% RSLogix 500 project Sauerstoff-Mess- und Kalibriersystem.RSS, saved by version 8.30.00.16 %
PROJECT "UNTITLED"    % processor: Bul.1763 MicroLogix 1100 Series B %

PROGRAM FILES
  LAD 2 "MAIN"  5 rungs
  LAD 3 "IO"  4 rungs
  LAD 4 "KALIBRIERU"  15 rungs

DATA FILES
  O0 OUTPUT  4 elements
  I1 INPUT  6 elements
  S2 STATUS  66 elements
  B3 BINARY  1 elements
  T4 TIMER  4 elements
  C5 COUNTER  1 elements
  R6 CONTROL  1 elements
  N7 INTEGER  9 elements
  F8 FLOAT  6 elements

LADDER 2 "MAIN"
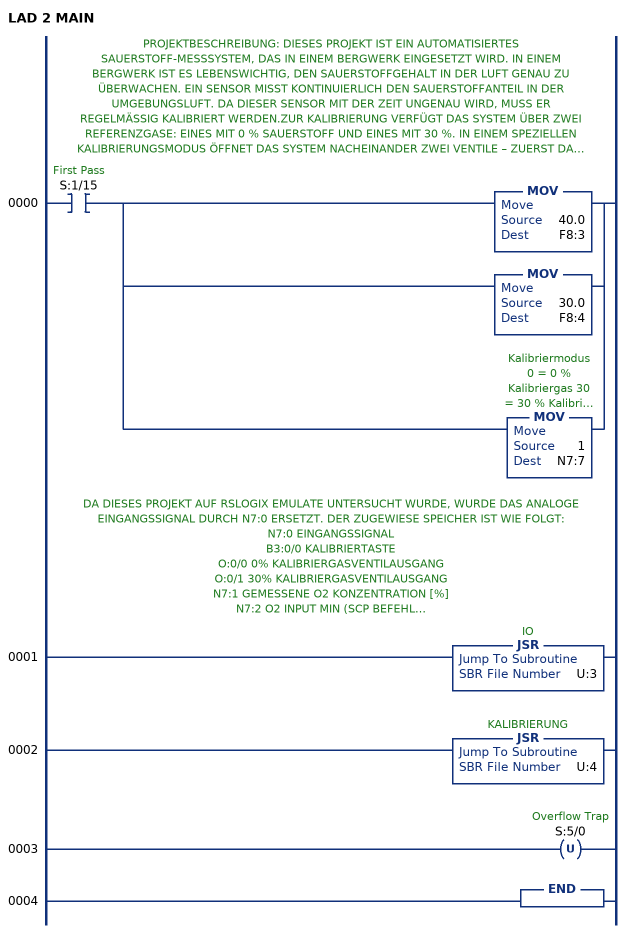
% Rung: 0 %
% PROJEKTBESCHREIBUNG: DIESES PROJEKT IST EIN AUTOMATISIERTES SAUERSTOFF-MESSSYSTEM, DAS IN EINEM BERGWERK EINGESETZT WIRD. IN EINEM BERGWERK IST ES LEBENSWICHTIG, DEN SAUERSTOFFGEHALT IN DER LUFT GENAU ZU ÜBERWACHEN. EIN SENSOR MISST KONTINUIERLICH DEN SAUERSTOFFANTEIL IN DER UMGEBUNGSLUFT. DA DIESER SENSOR MIT DER ZEIT UNGENAU WIRD, MUSS ER REGELMÄSSIG KALIBRIERT WERDEN.ZUR KALIBRIERUNG VERFÜGT DAS SYSTEM ÜBER ZWEI REFERENZGASE: EINES MIT 0 % SAUERSTOFF UND EINES MIT 30 %. IN EINEM SPEZIELLEN KALIBRIERUNGSMODUS ÖFFNET DAS SYSTEM NACHEINANDER ZWEI VENTILE – ZUERST DAS FÜR 0 %-GAS, DANN DAS FÜR 30 %-GAS – UND MISST JEWEILS 30 SEKUNDEN LANG DIE SENSORWERTE. AUS DIESEN MESSUNGEN BERECHNET DAS SYSTEM AUTOMATISCH KORREKTURWERTE, UM SPÄTERE SAUERSTOFFMESSUNGEN WIEDER KORREKT ANZEIGEN ZU KÖNNEN. %
SOR XIC S:1/15 BST MOV 40.0 F8:3 NXB MOV 30.0 F8:4 NXB MOV 1 N7:7 BND EOR
%   S:1/15  "First Pass" %
%   N7:7  "Kalibriermodus 0 = 0 % Kalibriergas 30 = 30 % Kalibriergas 1 = Idle Modus" %
% Rung: 1 %
% DA DIESES PROJEKT AUF RSLOGIX EMULATE UNTERSUCHT WURDE, WURDE DAS ANALOGE EINGANGSSIGNAL DURCH N7:0 ERSETZT. DER ZUGEWIESE SPEICHER IST WIE FOLGT:
% N7:0 EINGANGSSIGNAL
% B3:0/0 KALIBRIERTASTE
% O:0/0 0% KALIBRIERGASVENTILAUSGANG
% O:0/1 30% KALIBRIERGASVENTILAUSGANG
% N7:1 GEMESSENE O2 KONZENTRATION [%]
% N7:2 O2 INPUT MIN (SCP BEFEHL)
% N7:3 O2 INPUT MAX (SCP BEFEHL) %
SOR JSR U:3 EOR
%   U:3  "IO" %
% Rung: 2 %
SOR JSR U:4 EOR
%   U:4  "KALIBRIERUNG" %
% Rung: 3 %
SOR OTU S:5/0 EOR
%   S:5/0  "Overflow Trap" %
% Rung: 4 %
SOR END EOR

LADDER 3 "IO"
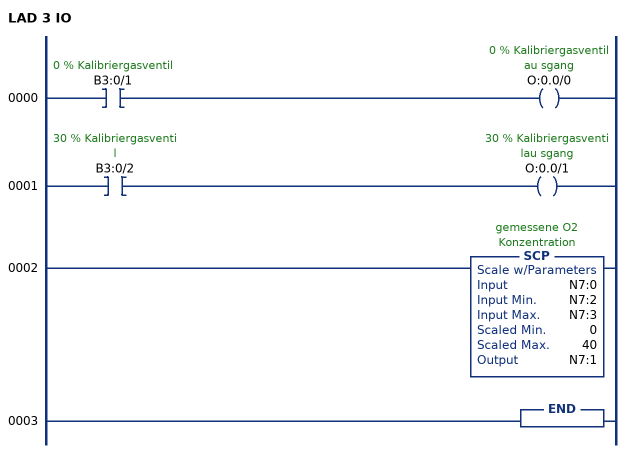
% Rung: 0 %
SOR XIC B3:0/1 OTE O:0.0/0 EOR
%   B3:0/1  "0 % Kalibriergasventil" %
%   O:0.0/0  "0 % Kalibriergasventilau sgang" %
% Rung: 1 %
SOR XIC B3:0/2 OTE O:0.0/1 EOR
%   B3:0/2  "30 % Kalibriergasventil" %
%   O:0.0/1  "30 % Kalibriergasventilau sgang" %
% Rung: 2 %
SOR SCP N7:0 N7:2 N7:3 0 40 N7:1 EOR
%   N7:0  "02 Eingangsignal" %
%   N7:2  "O2 Min" %
%   N7:3  "O2 Max" %
%   N7:1  "gemessene O2 Konzentration" %
% Rung: 3 %
SOR END EOR

LADDER 4 "KALIBRIERU"
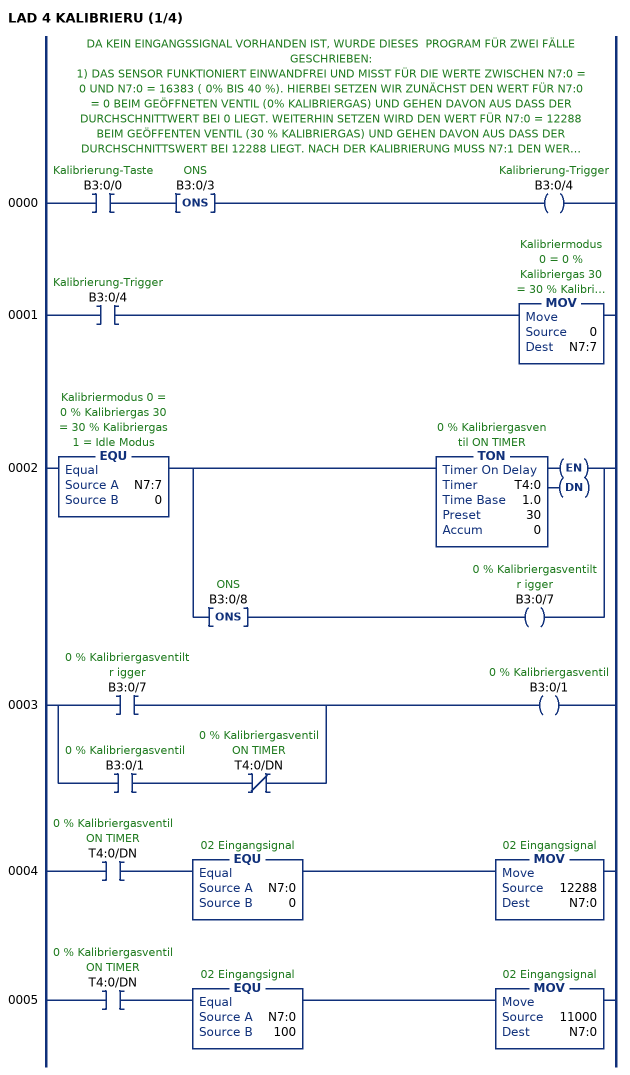
% Rung: 0 %
% DA KEIN EINGANGSSIGNAL VORHANDEN IST, WURDE DIESES  PROGRAM FÜR ZWEI FÄLLE GESCHRIEBEN:
% 1) DAS SENSOR FUNKTIONIERT EINWANDFREI UND MISST FÜR DIE WERTE ZWISCHEN N7:0 = 0 UND N7:0 = 16383 ( 0% BIS 40 %). HIERBEI SETZEN WIR ZUNÄCHST DEN WERT FÜR N7:0 = 0 BEIM GEÖFFNETEN VENTIL (0% KALIBRIERGAS) UND GEHEN DAVON AUS DASS DER DURCHSCHNITTWERT BEI 0 LIEGT. WEITERHIN SETZEN WIRD DEN WERT FÜR N7:0 = 12288 BEIM GEÖFFENTEN VENTIL (30 % KALIBRIERGAS) UND GEHEN DAVON AUS DASS DER DURCHSCHNITTSWERT BEI 12288 LIEGT. NACH DER KALIBRIERUNG MUSS N7:1 DEN WERT 30 ENTSPRECHEN (30%).
% 2) DAS SENSORWERTE WEICHEN AB. HIERBEI SETZEN WIR ZUNÄCHST DEN WERT FÜR N7:0 = 100 BEIM GEÖFFNETEN VENTIL (0% KALIBRIERGAS) UND GEHEN DAVON AUS DASS DER DURCHSCHNITTWERT BEI 100 LIEGT. WEITERHIN SETZEN WIRD DEN WERT FÜR N7:0 = 11000 BEIM GEÖFFENTEN VENTIL (30 % KALIBRIERGAS) UND GEHEN DAVON AUS DASS DER DURCHSCHNITTSWERT BEI 11000 LIEGT. NACH DER KALIBRIERUNG MUSS N7:1 DEN WERT 30 ENTSPRECHEN (30%).
% NACH JEDEM KALIBRIERVORGANG FINDET EINE ANPASSUNG (RECHNUNG AM ENDE) DER MIN OUTPUT UND MAX OUTPUT FÜR SCP BEFEHL %
SOR XIC B3:0/0 ONS B3:0/3 OTE B3:0/4 EOR
%   B3:0/0  "Kalibrierung-Taste" %
%   B3:0/3  "ONS" %
%   B3:0/4  "Kalibrierung-Trigger" %
% Rung: 1 %
SOR XIC B3:0/4 MOV 0 N7:7 EOR
%   B3:0/4  "Kalibrierung-Trigger" %
%   N7:7  "Kalibriermodus 0 = 0 % Kalibriergas 30 = 30 % Kalibriergas 1 = Idle Modus" %
% Rung: 2 %
SOR EQU N7:7 0 BST TON T4:0 1.0 30 0 NXB ONS B3:0/8 OTE B3:0/7 BND EOR
%   N7:7  "Kalibriermodus 0 = 0 % Kalibriergas 30 = 30 % Kalibriergas 1 = Idle Modus" %
%   T4:0  "0 % Kalibriergasventil ON TIMER" %
%   B3:0/8  "ONS" %
%   B3:0/7  "0 % Kalibriergasventiltr igger" %
% Rung: 3 %
SOR BST XIC B3:0/7 NXB XIC B3:0/1 XIO T4:0/DN BND OTE B3:0/1 EOR
%   B3:0/7  "0 % Kalibriergasventiltr igger" %
%   B3:0/1  "0 % Kalibriergasventil" %
%   T4:0  "0 % Kalibriergasventil ON TIMER" %
% Rung: 4 %
SOR XIC T4:0/DN EQU N7:0 0 MOV 12288 N7:0 EOR
%   T4:0  "0 % Kalibriergasventil ON TIMER" %
%   N7:0  "02 Eingangsignal" %
% Rung: 5 %
SOR XIC T4:0/DN EQU N7:0 100 MOV 11000 N7:0 EOR
%   T4:0  "0 % Kalibriergasventil ON TIMER" %
%   N7:0  "02 Eingangsignal" %

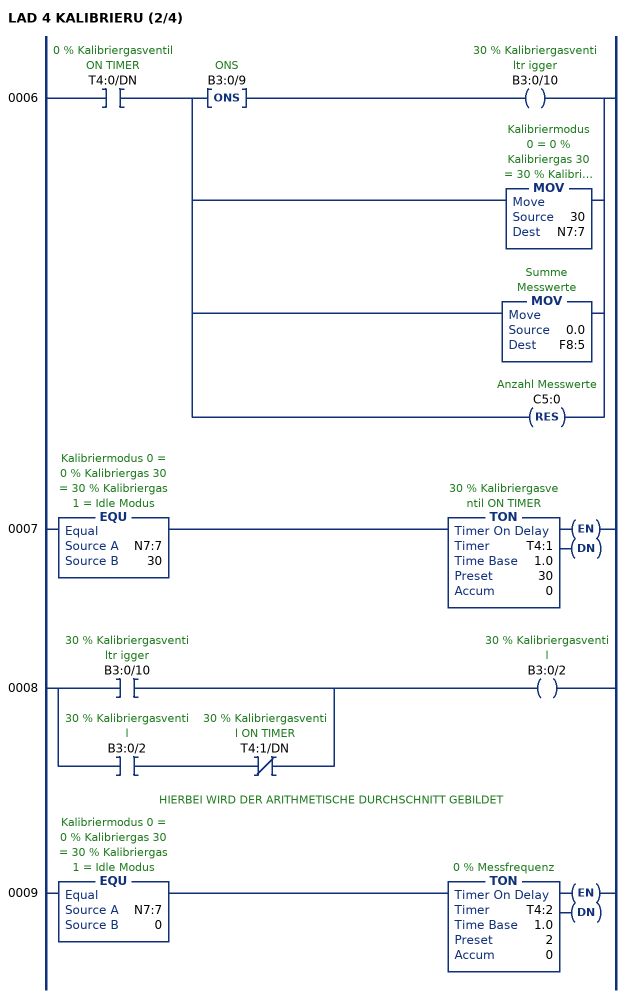
% Rung: 6 %
SOR XIC T4:0/DN BST ONS B3:0/9 OTE B3:0/10 NXB MOV 30 N7:7 NXB MOV 0.0 F8:5 NXB RES C5:0 BND EOR
%   T4:0  "0 % Kalibriergasventil ON TIMER" %
%   B3:0/9  "ONS" %
%   B3:0/10  "30 % Kalibriergasventiltr igger" %
%   N7:7  "Kalibriermodus 0 = 0 % Kalibriergas 30 = 30 % Kalibriergas 1 = Idle Modus" %
%   F8:5  "Summe Messwerte" %
%   C5:0  "Anzahl Messwerte" %
% Rung: 7 %
SOR EQU N7:7 30 TON T4:1 1.0 30 0 EOR
%   N7:7  "Kalibriermodus 0 = 0 % Kalibriergas 30 = 30 % Kalibriergas 1 = Idle Modus" %
%   T4:1  "30 % Kalibriergasventil ON TIMER" %
% Rung: 8 %
SOR BST XIC B3:0/10 NXB XIC B3:0/2 XIO T4:1/DN BND OTE B3:0/2 EOR
%   B3:0/10  "30 % Kalibriergasventiltr igger" %
%   B3:0/2  "30 % Kalibriergasventil" %
%   T4:1  "30 % Kalibriergasventil ON TIMER" %
% Rung: 9 %
% HIERBEI WIRD DER ARITHMETISCHE DURCHSCHNITT GEBILDET %
SOR EQU N7:7 0 TON T4:2 1.0 2 0 EOR
%   N7:7  "Kalibriermodus 0 = 0 % Kalibriergas 30 = 30 % Kalibriergas 1 = Idle Modus" %
%   T4:2  "0 % Messfrequenz" %

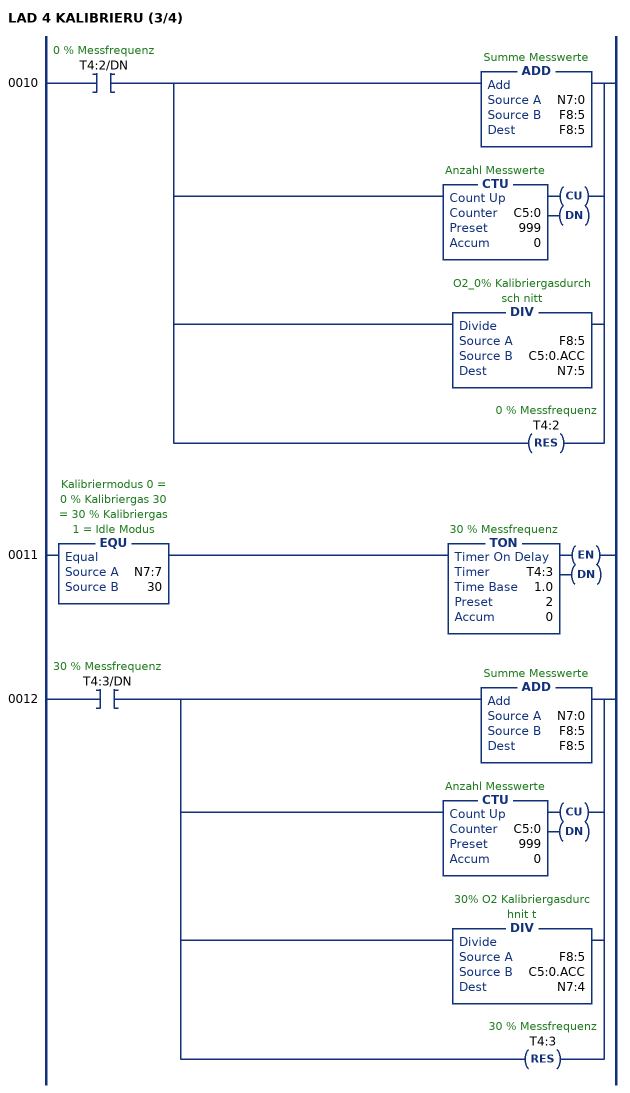
% Rung: 10 %
SOR XIC T4:2/DN BST ADD N7:0 F8:5 F8:5 NXB CTU C5:0 999 0 NXB DIV F8:5 C5:0.ACC N7:5 NXB RES T4:2 BND EOR
%   T4:2  "0 % Messfrequenz" %
%   N7:0  "02 Eingangsignal" %
%   F8:5  "Summe Messwerte" %
%   C5:0  "Anzahl Messwerte" %
%   N7:5  "O2_0% Kalibriergasdurchsch nitt" %
% Rung: 11 %
SOR EQU N7:7 30 TON T4:3 1.0 2 0 EOR
%   N7:7  "Kalibriermodus 0 = 0 % Kalibriergas 30 = 30 % Kalibriergas 1 = Idle Modus" %
%   T4:3  "30 % Messfrequenz" %
% Rung: 12 %
SOR XIC T4:3/DN BST ADD N7:0 F8:5 F8:5 NXB CTU C5:0 999 0 NXB DIV F8:5 C5:0.ACC N7:4 NXB RES T4:3 BND EOR
%   T4:3  "30 % Messfrequenz" %
%   N7:0  "02 Eingangsignal" %
%   F8:5  "Summe Messwerte" %
%   C5:0  "Anzahl Messwerte" %
%   N7:4  "30% O2 Kalibriergasdurchnit t" %

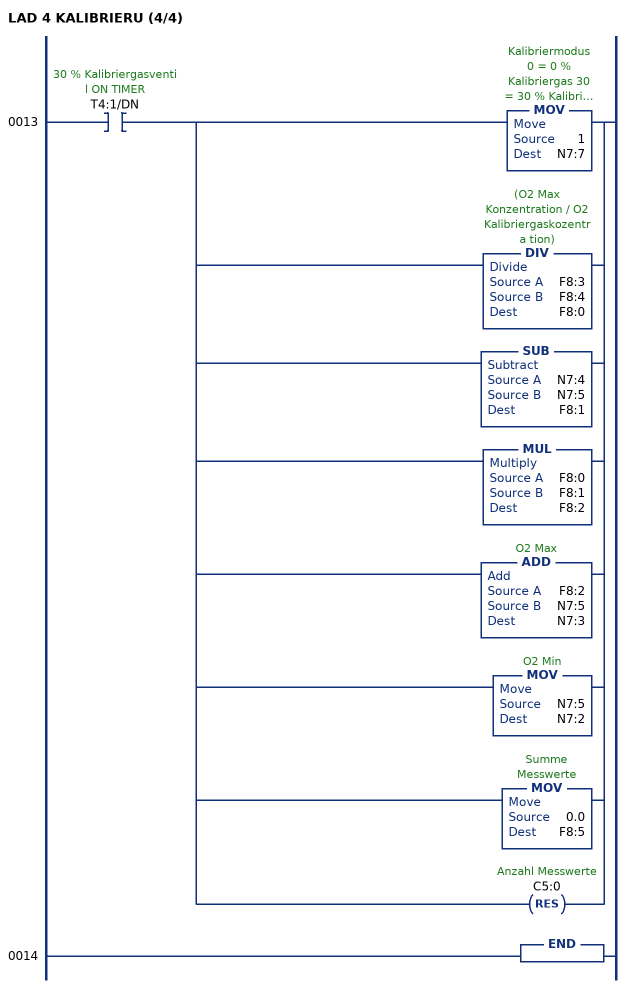
% Rung: 13 %
SOR XIC T4:1/DN BST MOV 1 N7:7 NXB DIV F8:3 F8:4 F8:0 NXB SUB N7:4 N7:5 F8:1 NXB MUL F8:0 F8:1 F8:2 NXB ADD F8:2 N7:5 N7:3 NXB MOV N7:5 N7:2 NXB MOV 0.0 F8:5 NXB RES C5:0 BND EOR
%   T4:1  "30 % Kalibriergasventil ON TIMER" %
%   N7:7  "Kalibriermodus 0 = 0 % Kalibriergas 30 = 30 % Kalibriergas 1 = Idle Modus" %
%   F8:0  "(O2 Max Konzentration / O2 Kalibriergaskozentra tion)" %
%   N7:4  "30% O2 Kalibriergasdurchnit t" %
%   N7:5  "O2_0% Kalibriergasdurchsch nitt" %
%   N7:3  "O2 Max" %
%   N7:2  "O2 Min" %
%   F8:5  "Summe Messwerte" %
%   C5:0  "Anzahl Messwerte" %
% Rung: 14 %
SOR END EOR

OTHER DOCUMENTED ADDRESSES
  B3:0/5  "Kalibrierung"
  B3:0/6  "Kalibrierung- Interrupt"
  B3:0/11  "ONS"
  B3:0/12  "ONS"
  N7:6  "Input Max"
  N7:8  "Summe Messwerte"
  U:5  "Kalibrierungsrechnun g"

COMMENTS NOT ATTACHED TO A CURRENT RUNG
  U:3: DA DIESES PROJEKT AUF RSLOGIX EMULATE UNTERSUCHT WURDE, WURDE DAS ANALOGE EINGANGSSIGNAL DURCH N7:0 ERSETZT. DER ZUGEWIESE SPEICHER IST WIE FOLGT:
    N7:0 EINGANGSSIGNAL
    B3:0/0 KALIBRIERTASTE
    O:0/0 0% KALIBRIERGASVENTILAUSGANG
    O:0/1 30% KALIBRIERGASVENTILAUSGANG
    N7:1 GEMESSENE O2 KONZENTRATION [%]
    N7:2 O2 INPUT MIN (SCP BEFEHL)
    N7:3 O2 INPUT MAX (SCP BEFEHL)

DATA TABLE (non-zero values as saved)
DATA T4
% .PRE .ACC %
% T4:0 % 30 0
% T4:1 % 30 0
% T4:2 % 2 0
% T4:3 % 2 0
DATA C5
% .PRE .ACC %
% C5:0 % 999 0
